// TIA Portal V15.1 export
// export: Created 2020-06-12T07:35:51.7099609Z, ExportSetting None, DisplayName Totally Integrated Automation Portal, DisplayVersion V15.1, DisplayName TIA Portal Openness, DisplayVersion V15.1, DisplayName STEP 7 Professional, DisplayVersion V15.1, DisplayName STEP 7 Safety, DisplayVersion V15.1, DisplayName WinCC Advanced, DisplayVersion V15.1
FUNCTION "MELT_Slag" : Void   // FC132, FBD
{ S7_Optimized_Access := 'TRUE' }
// stored: SetENOAutomatically False
   VAR_TEMP
      tStartAmount : Real;
      tReqDummy : Bool;
      tReqPrepare : Bool;
      tReqManFilled : Bool;
      tReqCancel : Bool;
      tReqReset : Bool;
      tSSIsLoaded : Bool;
      tPreBaseSlag : Bool;
      tDoBaseLoad : Bool;
      tBSIsLoaded : Bool;
      tReqBaseLoad : Bool;
      tReset : Bool;
      tBaseAmount : Real;
      tFeedingTime : Real;
      tIdx : Int;
      tStartTime : Real;
      tWeightDiff : Real;
      tDurationDiff : Real;
   END_VAR
   VAR_TEMP   // added for the SCL form of the ladder/FBD networks
      _w1 : Bool;
      _w2 : Bool;
   END_VAR
BEGIN

REGION Network 1: HMI Request
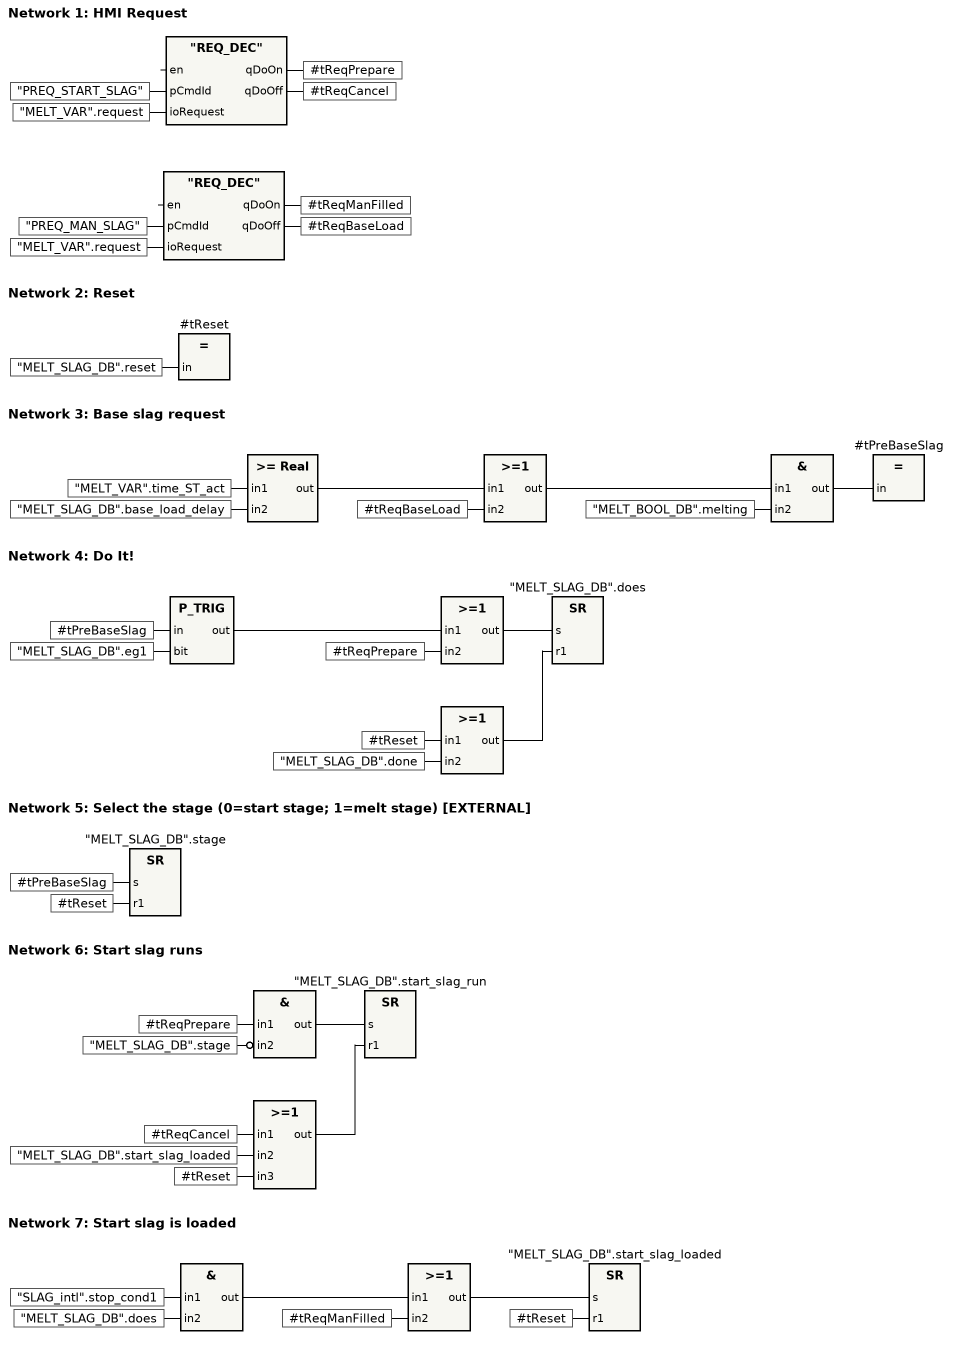
   "REQ_DEC"(pCmdId := "PREQ_START_SLAG",
             ioRequest := "MELT_VAR".request,
             qDoOn => #tReqPrepare,
             qDoOff => #tReqCancel);
   "REQ_DEC"(pCmdId := "PREQ_MAN_SLAG",
             ioRequest := "MELT_VAR".request,
             qDoOn => #tReqManFilled,
             qDoOff => #tReqBaseLoad);
END_REGION

REGION Network 2: Reset
   #tReset := "MELT_SLAG_DB".reset;
END_REGION

REGION Network 3: Base slag request
   #tPreBaseSlag := (("MELT_VAR".time_ST_act >= "MELT_SLAG_DB".base_load_delay) OR #tReqBaseLoad) AND "MELT_BOOL_DB".melting;
END_REGION

REGION Network 4: Do It!
   #_w1 := #tPreBaseSlag AND NOT "MELT_SLAG_DB".eg1;   // rising edge
   "MELT_SLAG_DB".eg1 := #tPreBaseSlag;
   IF #_w1 OR #tReqPrepare THEN
       "MELT_SLAG_DB".does := TRUE;   // SR flip-flop
   END_IF;
   IF #tReset OR "MELT_SLAG_DB".done THEN "MELT_SLAG_DB".does := FALSE; END_IF;
END_REGION

REGION Network 5: Select the stage (0=start stage; 1=melt stage) [EXTERNAL]
   IF #tPreBaseSlag THEN
       "MELT_SLAG_DB".stage := TRUE;   // SR flip-flop
   END_IF;
   IF #tReset THEN "MELT_SLAG_DB".stage := FALSE; END_IF;
END_REGION

REGION Network 6: Start slag runs
   IF #tReqPrepare AND NOT "MELT_SLAG_DB".stage THEN
       "MELT_SLAG_DB".start_slag_run := TRUE;   // SR flip-flop
   END_IF;
   IF #tReqCancel OR "MELT_SLAG_DB".start_slag_loaded OR #tReset THEN
       "MELT_SLAG_DB".start_slag_run := FALSE;
   END_IF;
END_REGION

REGION Network 7: Start slag is loaded
   IF ("SLAG_intl".stop_cond1 AND "MELT_SLAG_DB".does) OR #tReqManFilled THEN
       "MELT_SLAG_DB".start_slag_loaded := TRUE;   // SR flip-flop
   END_IF;
   IF #tReset THEN "MELT_SLAG_DB".start_slag_loaded := FALSE; END_IF;
END_REGION

REGION Network 8: Base slag runs
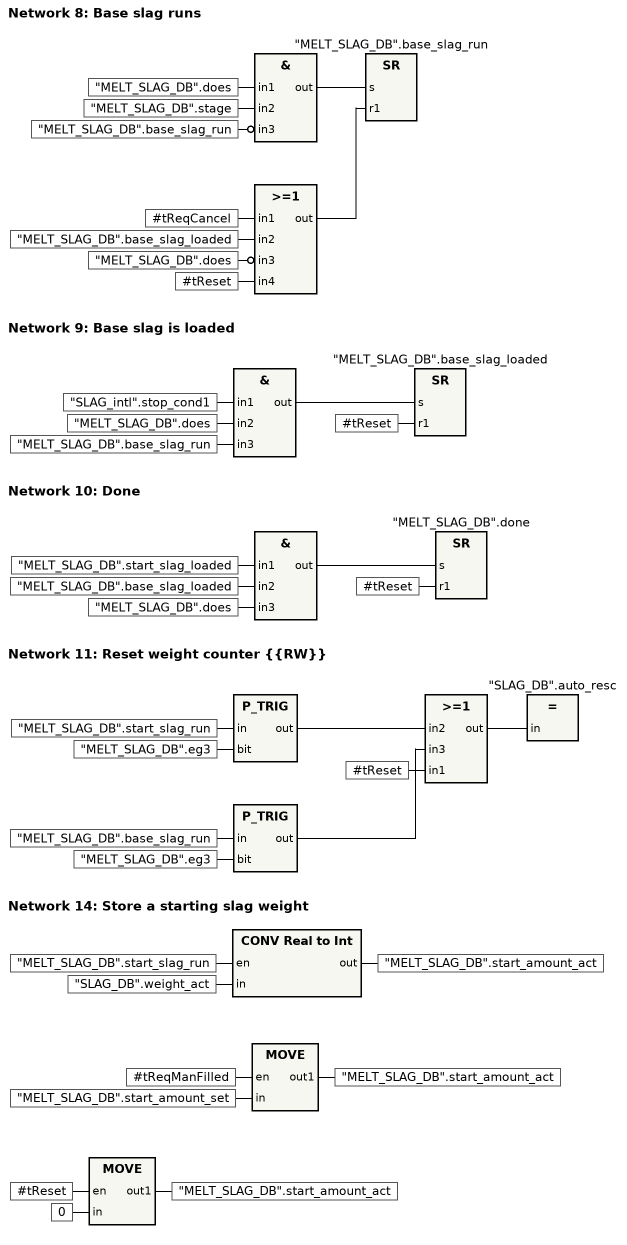
   IF "MELT_SLAG_DB".does AND "MELT_SLAG_DB".stage AND NOT "MELT_SLAG_DB".base_slag_run THEN
       "MELT_SLAG_DB".base_slag_run := TRUE;   // SR flip-flop
   END_IF;
   IF #tReqCancel OR "MELT_SLAG_DB".base_slag_loaded OR NOT "MELT_SLAG_DB".does OR #tReset THEN
       "MELT_SLAG_DB".base_slag_run := FALSE;
   END_IF;
END_REGION

REGION Network 9: Base slag is loaded
   IF "SLAG_intl".stop_cond1 AND "MELT_SLAG_DB".does AND "MELT_SLAG_DB".base_slag_run THEN
       "MELT_SLAG_DB".base_slag_loaded := TRUE;   // SR flip-flop
   END_IF;
   IF #tReset THEN "MELT_SLAG_DB".base_slag_loaded := FALSE; END_IF;
END_REGION

REGION Network 10: Done
   IF "MELT_SLAG_DB".start_slag_loaded AND "MELT_SLAG_DB".base_slag_loaded AND "MELT_SLAG_DB".does THEN
       "MELT_SLAG_DB".done := TRUE;   // SR flip-flop
   END_IF;
   IF #tReset THEN "MELT_SLAG_DB".done := FALSE; END_IF;
END_REGION

REGION Network 11: Reset weight counter {{RW}}
   #_w1 := "MELT_SLAG_DB".start_slag_run AND NOT "MELT_SLAG_DB".eg3;   // rising edge
   "MELT_SLAG_DB".eg3 := "MELT_SLAG_DB".start_slag_run;
   #_w2 := "MELT_SLAG_DB".base_slag_run AND NOT "MELT_SLAG_DB".eg3;   // rising edge
   "MELT_SLAG_DB".eg3 := "MELT_SLAG_DB".base_slag_run;
   "SLAG_DB".auto_resc := #_w1 OR #_w2 OR #tReset;
END_REGION

REGION Network 12 (SCL): Calculation slag weight and base weight
   "MELT_SLAG_DB".base_amount_set := "MELT_SLAG_DB".tot_amount_set - "MELT_SLAG_DB".start_amount_set;
   CASE "MELT_SLAG_DB".cm OF
       1:
           "MELT_SLAG_DB".base_slag_rate := "MELT_SLAG_DB".base_amount_set / "MELT_SLAG_DB".base_load_time_set;
       2:  (*
           #tWeightDiff := ("MELT_SLAG_DB".base_amount_set - "MELT_SLAG_DB".base_amount_act);
           #tDurationDiff := ("MELT_SLAG_DB".base_load_time_set - "MELT_SLAG_DB".base_load_time_act);
           "MELT_SLAG_DB".base_slag_rate := #tWeightDiff / #tDurationDiff;
           *);
       ELSE
           ;
   END_CASE;
END_REGION

REGION Network 13 (SCL): Setpoints
   IF "MELT_SLAG_DB".start_slag_run THEN
       "SLAG_DB".weight_set := "MELT_SLAG_DB".start_amount_set;
       "SLAG_DB".feed_rate_set := 50.0;
   ELSIF "MELT_SLAG_DB".base_slag_run THEN
       "SLAG_DB".weight_set := "MELT_SLAG_DB".base_amount_set;
       "SLAG_DB".feed_rate_set := "MELT_SLAG_DB".base_slag_rate;
   END_IF;
END_REGION

REGION Network 14: Store a starting slag weight
   IF "MELT_SLAG_DB".start_slag_run THEN
       "MELT_SLAG_DB".start_amount_act := REAL_TO_INT("SLAG_DB".weight_act);
   END_IF;
   IF #tReqManFilled THEN "MELT_SLAG_DB".start_amount_act := "MELT_SLAG_DB".start_amount_set; END_IF;
   IF #tReset THEN "MELT_SLAG_DB".start_amount_act := 0; END_IF;
END_REGION

REGION Network 15: Store a base slag weight
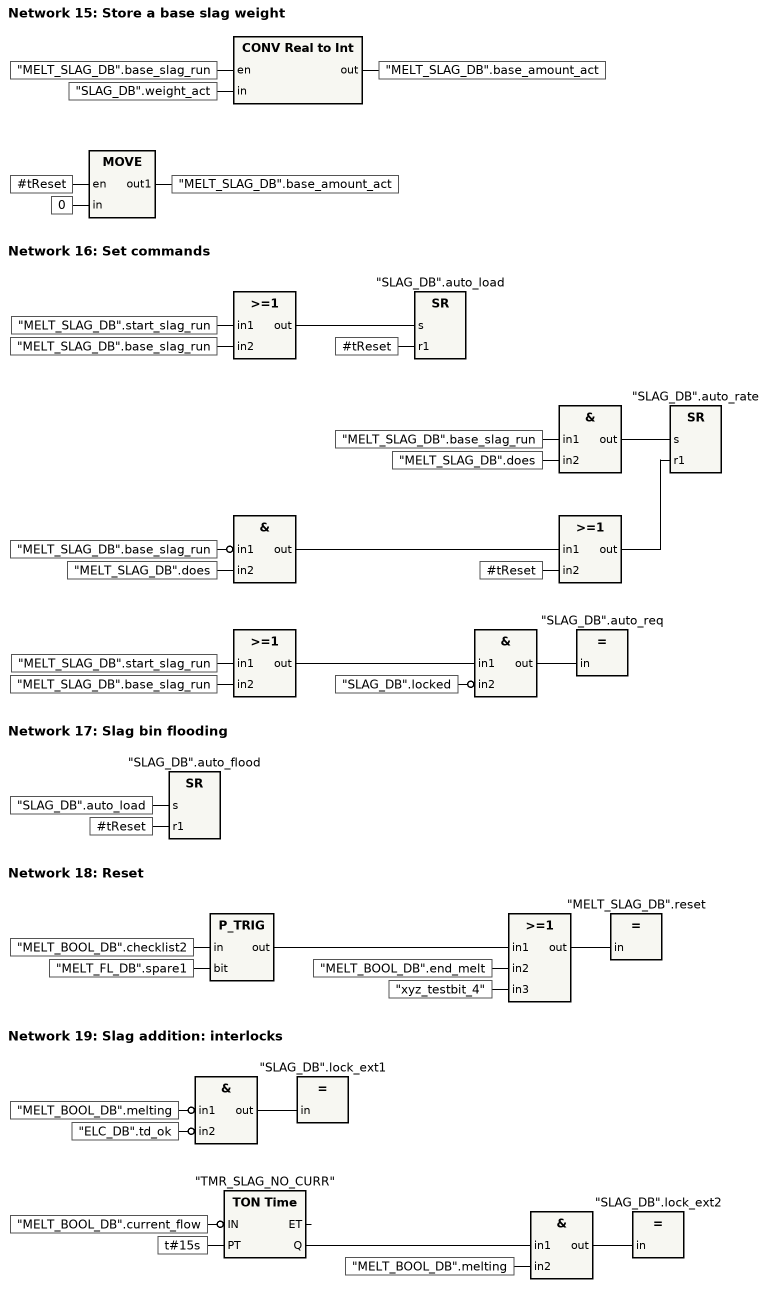
   IF "MELT_SLAG_DB".base_slag_run THEN
       "MELT_SLAG_DB".base_amount_act := REAL_TO_INT("SLAG_DB".weight_act);
   END_IF;
   IF #tReset THEN "MELT_SLAG_DB".base_amount_act := 0; END_IF;
END_REGION

REGION Network 16: Set commands
   IF "MELT_SLAG_DB".start_slag_run OR "MELT_SLAG_DB".base_slag_run THEN
       "SLAG_DB".auto_load := TRUE;   // SR flip-flop
   END_IF;
   IF #tReset THEN "SLAG_DB".auto_load := FALSE; END_IF;
   IF "MELT_SLAG_DB".base_slag_run AND "MELT_SLAG_DB".does THEN
       "SLAG_DB".auto_rate := TRUE;   // SR flip-flop
   END_IF;
   IF (NOT "MELT_SLAG_DB".base_slag_run AND "MELT_SLAG_DB".does) OR #tReset THEN
       "SLAG_DB".auto_rate := FALSE;
   END_IF;
   "SLAG_DB".auto_req := ("MELT_SLAG_DB".start_slag_run OR "MELT_SLAG_DB".base_slag_run) AND NOT "SLAG_DB".locked;
END_REGION

REGION Network 17: Slag bin flooding
   IF "SLAG_DB".auto_load THEN
       "SLAG_DB".auto_flood := TRUE;   // SR flip-flop
   END_IF;
   IF #tReset THEN "SLAG_DB".auto_flood := FALSE; END_IF;
END_REGION

REGION Network 18: Reset
   #_w1 := "MELT_BOOL_DB".checklist2 AND NOT "MELT_FL_DB".spare1;   // rising edge
   "MELT_FL_DB".spare1 := "MELT_BOOL_DB".checklist2;
   "MELT_SLAG_DB".reset := #_w1 OR "MELT_BOOL_DB".end_melt OR "xyz_testbit_4";
END_REGION

REGION Network 19: Slag addition: interlocks
   "SLAG_DB".lock_ext1 := NOT "MELT_BOOL_DB".melting AND NOT "ELC_DB".td_ok;
   "TMR_SLAG_NO_CURR".TON(IN := NOT "MELT_BOOL_DB".current_flow, PT := t#15s);
   "SLAG_DB".lock_ext2 := "TMR_SLAG_NO_CURR".Q AND "MELT_BOOL_DB".melting;
END_REGION

REGION Network 20: HMI status
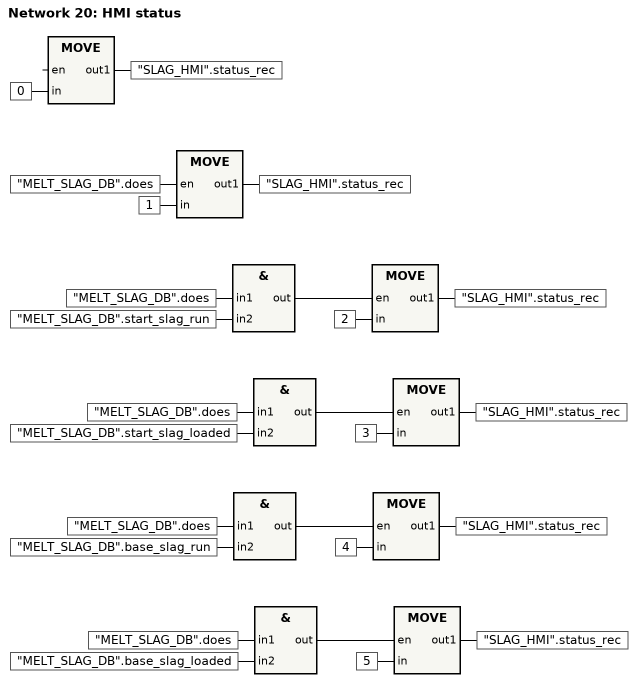
   "SLAG_HMI".status_rec := 0;
   IF "MELT_SLAG_DB".does THEN "SLAG_HMI".status_rec := 1; END_IF;
   IF "MELT_SLAG_DB".does AND "MELT_SLAG_DB".start_slag_run THEN "SLAG_HMI".status_rec := 2; END_IF;
   IF "MELT_SLAG_DB".does AND "MELT_SLAG_DB".start_slag_loaded THEN "SLAG_HMI".status_rec := 3; END_IF;
   IF "MELT_SLAG_DB".does AND "MELT_SLAG_DB".base_slag_run THEN "SLAG_HMI".status_rec := 4; END_IF;
   IF "MELT_SLAG_DB".does AND "MELT_SLAG_DB".base_slag_loaded THEN "SLAG_HMI".status_rec := 5; END_IF;
END_REGION

REGION Network 21 (SCL): HMI status: progress
   "MELT_SLAG_DB".progress := INT_TO_REAL("MELT_SLAG_DB".base_amount_act) / INT_TO_REAL("MELT_SLAG_DB".base_amount_set) * 100;
END_REGION

REGION Network 22 (SCL): HMI status: time
   IF "MELT_SLAG_DB".base_slag_run THEN
       "MELT_SLAG_DB".base_load_time_act := "MELT_VAR".time_ST_act - "MELT_SLAG_DB".base_load_delay;
   END_IF;
   IF "MELT_SLAG_DB".start_slag_run THEN
       "MELT_SLAG_DB".base_load_time_act := 0;
   END_IF;
END_REGION

REGION Network 23: [[END]]
END_REGION
END_FUNCTION
